// TIA Portal V19 export
FUNCTION_BLOCK "Sensors"   // FB4, LAD
{ S7_Optimized_Access := 'TRUE' }
// stored: MemoryReserve 100, SetENOAutomatically false
   VAR
      GenericSensor11 { S7_SetPoint := 'True'} : "GenericSensor";
      GenericSensor12 { S7_SetPoint := 'True'} : "GenericSensor";
      GenericSensor13 { S7_SetPoint := 'True'} : "GenericSensor";
      GenericSensor21 { S7_SetPoint := 'True'} : "GenericSensor";
      GenericSensor22 { S7_SetPoint := 'True'} : "GenericSensor";
      PubJsonMqttInst11 { S7_SetPoint := 'True'} : "PublishJsonMqtt";
      PubJsonMqttInst12 { S7_SetPoint := 'True'} : "PublishJsonMqtt";
      PubJsonMqttInst13 { S7_SetPoint := 'True'} : "PublishJsonMqtt";
      PubJsonMqttInst21 { S7_SetPoint := 'True'} : "PublishJsonMqtt";
      PubJsonMqttInst22 { S7_SetPoint := 'True'} : "PublishJsonMqtt";
      tpGen01 { S7_SetPoint := 'True'} : TP_TIME;
      tpGen02 { S7_SetPoint := 'True'} : TP_TIME;
      tpGen03 { S7_SetPoint := 'True'} : TP_TIME;
      tpGen04 { S7_SetPoint := 'True'} : TP_TIME;
   END_VAR
   VAR_TEMP
      Sensor11 : Real;
      Sensor12 : Real;
      Sensor13 : Real;
      Sensor21 : Real;
      Sensor22 : Real;
   END_VAR
   VAR_TEMP   // added for the SCL form of the ladder/FBD networks
      _w1 : Bool;
   END_VAR
BEGIN

REGION Network 1 (SCL): Generator for data publish Machine 1
   // Define how often sensors are polled and mqtt data sent.
   #tpGen01(IN:=NOT #tpGen02.Q,
            PT:=T#1S);

   #tpGen02(IN:=NOT #tpGen01.Q,
            PT:=T#50MS);
END_REGION

REGION Network 2 (SCL): Generator for data publish Machine 2
   #tpGen03(IN := NOT #tpGen04.Q,
            PT := T#3S);

   #tpGen04(IN := NOT #tpGen03.Q,
            PT := T#50MS);
END_REGION

REGION Network 3: Line 1 / Machine 1 / Sensor 001
   // SELECTOR defines if simulated sensor value or real IO-Link sensor value is evaluated and published by MQTT.
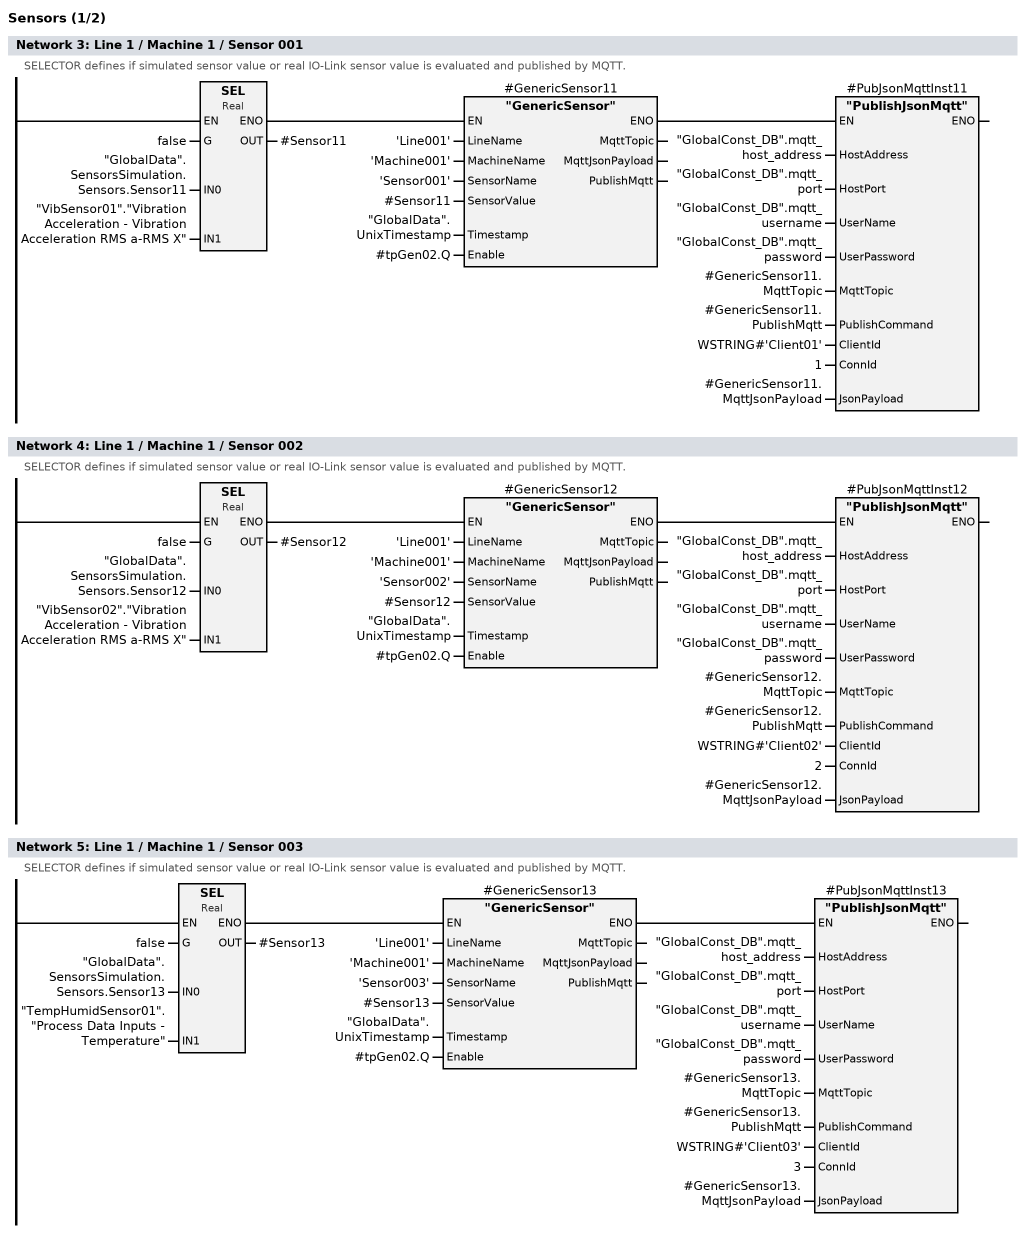
   RUNG wire#powerrail
      { S7_Templates := "value_type := Real" } SEL(g := false, in0 := "GlobalData".SensorsSimulation.Sensors.Sensor11, in1 := "VibSensor01"."Vibration Acceleration - Vibration Acceleration RMS a-RMS X", out => #Sensor11)
      #GenericSensor11(LineName := 'Line001', MachineName := 'Machine001', SensorName := 'Sensor001', SensorValue := #Sensor11, Timestamp := "GlobalData".UnixTimestamp, Enable := #tpGen02.Q, MqttTopic =>, MqttJsonPayload =>, PublishMqtt =>)
      #PubJsonMqttInst11(HostAddress := "GlobalConst_DB".mqtt_host_address, HostPort := "GlobalConst_DB".mqtt_port, UserName := "GlobalConst_DB".mqtt_username, UserPassword := "GlobalConst_DB".mqtt_password, MqttTopic := #GenericSensor11.MqttTopic, PublishCommand := #GenericSensor11.PublishMqtt, ClientId := WSTRING#'Client01', ConnId := 1, JsonPayload := #GenericSensor11.MqttJsonPayload)
   END_RUNG
   // the same network as SCL:
   // ENO of a box is taken as its EN; it also drops when the box reports an error
   #Sensor11 := SEL(G := false, IN0 := "GlobalData".SensorsSimulation.Sensors.Sensor11, IN1 := "VibSensor01"."Vibration Acceleration - Vibration Acceleration RMS a-RMS X");
   #GenericSensor11(LineName := 'Line001',   // "GenericSensor"
                    MachineName := 'Machine001',
                    SensorName := 'Sensor001',
                    SensorValue := #Sensor11,
                    Timestamp := "GlobalData".UnixTimestamp,
                    Enable := #tpGen02.Q,
                    ENO => #_w1);
   IF #_w1 THEN
       #PubJsonMqttInst11(HostAddress := "GlobalConst_DB".mqtt_host_address,   // "PublishJsonMqtt"
                          HostPort := "GlobalConst_DB".mqtt_port,
                          UserName := "GlobalConst_DB".mqtt_username,
                          UserPassword := "GlobalConst_DB".mqtt_password,
                          MqttTopic := #GenericSensor11.MqttTopic,
                          PublishCommand := #GenericSensor11.PublishMqtt,
                          ClientId := WSTRING#'Client01',
                          ConnId := 1,
                          JsonPayload := #GenericSensor11.MqttJsonPayload);
   END_IF;
END_REGION

REGION Network 4: Line 1 / Machine 1 / Sensor 002
   // SELECTOR defines if simulated sensor value or real IO-Link sensor value is evaluated and published by MQTT.
   RUNG wire#powerrail
      { S7_Templates := "value_type := Real" } SEL(g := false, in0 := "GlobalData".SensorsSimulation.Sensors.Sensor12, in1 := "VibSensor02"."Vibration Acceleration - Vibration Acceleration RMS a-RMS X", out => #Sensor12)
      #GenericSensor12(LineName := 'Line001', MachineName := 'Machine001', SensorName := 'Sensor002', SensorValue := #Sensor12, Timestamp := "GlobalData".UnixTimestamp, Enable := #tpGen02.Q, MqttTopic =>, MqttJsonPayload =>, PublishMqtt =>)
      #PubJsonMqttInst12(HostAddress := "GlobalConst_DB".mqtt_host_address, HostPort := "GlobalConst_DB".mqtt_port, UserName := "GlobalConst_DB".mqtt_username, UserPassword := "GlobalConst_DB".mqtt_password, MqttTopic := #GenericSensor12.MqttTopic, PublishCommand := #GenericSensor12.PublishMqtt, ClientId := WSTRING#'Client02', ConnId := 2, JsonPayload := #GenericSensor12.MqttJsonPayload)
   END_RUNG
   // the same network as SCL:
   // ENO of a box is taken as its EN; it also drops when the box reports an error
   #Sensor12 := SEL(G := false, IN0 := "GlobalData".SensorsSimulation.Sensors.Sensor12, IN1 := "VibSensor02"."Vibration Acceleration - Vibration Acceleration RMS a-RMS X");
   #GenericSensor12(LineName := 'Line001',   // "GenericSensor"
                    MachineName := 'Machine001',
                    SensorName := 'Sensor002',
                    SensorValue := #Sensor12,
                    Timestamp := "GlobalData".UnixTimestamp,
                    Enable := #tpGen02.Q,
                    ENO => #_w1);
   IF #_w1 THEN
       #PubJsonMqttInst12(HostAddress := "GlobalConst_DB".mqtt_host_address,   // "PublishJsonMqtt"
                          HostPort := "GlobalConst_DB".mqtt_port,
                          UserName := "GlobalConst_DB".mqtt_username,
                          UserPassword := "GlobalConst_DB".mqtt_password,
                          MqttTopic := #GenericSensor12.MqttTopic,
                          PublishCommand := #GenericSensor12.PublishMqtt,
                          ClientId := WSTRING#'Client02',
                          ConnId := 2,
                          JsonPayload := #GenericSensor12.MqttJsonPayload);
   END_IF;
END_REGION

REGION Network 5: Line 1 / Machine 1 / Sensor 003
   // SELECTOR defines if simulated sensor value or real IO-Link sensor value is evaluated and published by MQTT.
   RUNG wire#powerrail
      { S7_Templates := "value_type := Real" } SEL(g := false, in0 := "GlobalData".SensorsSimulation.Sensors.Sensor13, in1 := "TempHumidSensor01"."Process Data Inputs - Temperature", out => #Sensor13)
      #GenericSensor13(LineName := 'Line001', MachineName := 'Machine001', SensorName := 'Sensor003', SensorValue := #Sensor13, Timestamp := "GlobalData".UnixTimestamp, Enable := #tpGen02.Q, MqttTopic =>, MqttJsonPayload =>, PublishMqtt =>)
      #PubJsonMqttInst13(HostAddress := "GlobalConst_DB".mqtt_host_address, HostPort := "GlobalConst_DB".mqtt_port, UserName := "GlobalConst_DB".mqtt_username, UserPassword := "GlobalConst_DB".mqtt_password, MqttTopic := #GenericSensor13.MqttTopic, PublishCommand := #GenericSensor13.PublishMqtt, ClientId := WSTRING#'Client03', ConnId := 3, JsonPayload := #GenericSensor13.MqttJsonPayload)
   END_RUNG
   // the same network as SCL:
   // ENO of a box is taken as its EN; it also drops when the box reports an error
   #Sensor13 := SEL(G := false, IN0 := "GlobalData".SensorsSimulation.Sensors.Sensor13, IN1 := "TempHumidSensor01"."Process Data Inputs - Temperature");
   #GenericSensor13(LineName := 'Line001',   // "GenericSensor"
                    MachineName := 'Machine001',
                    SensorName := 'Sensor003',
                    SensorValue := #Sensor13,
                    Timestamp := "GlobalData".UnixTimestamp,
                    Enable := #tpGen02.Q,
                    ENO => #_w1);
   IF #_w1 THEN
       #PubJsonMqttInst13(HostAddress := "GlobalConst_DB".mqtt_host_address,   // "PublishJsonMqtt"
                          HostPort := "GlobalConst_DB".mqtt_port,
                          UserName := "GlobalConst_DB".mqtt_username,
                          UserPassword := "GlobalConst_DB".mqtt_password,
                          MqttTopic := #GenericSensor13.MqttTopic,
                          PublishCommand := #GenericSensor13.PublishMqtt,
                          ClientId := WSTRING#'Client03',
                          ConnId := 3,
                          JsonPayload := #GenericSensor13.MqttJsonPayload);
   END_IF;
END_REGION

REGION Network 6: Line 1 / Machine 2 / Sensor 001
   // SELECTOR defines if simulated sensor value or real IO-Link sensor value is evaluated and published by MQTT.
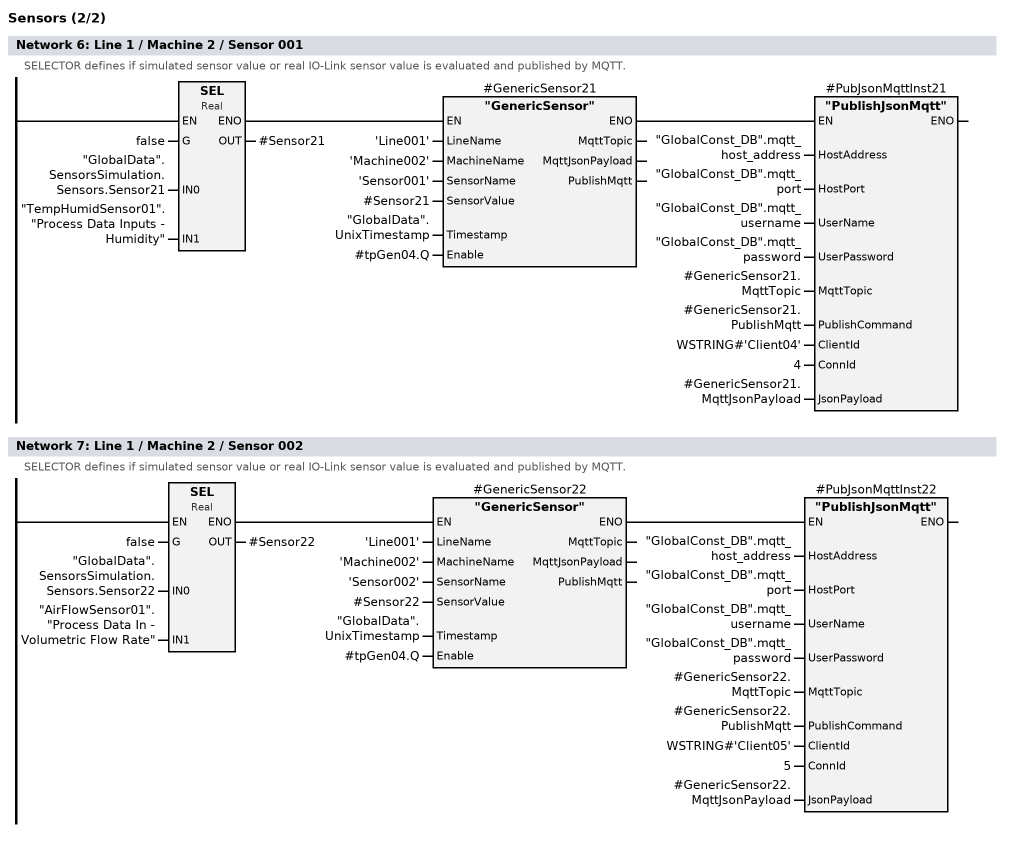
   RUNG wire#powerrail
      { S7_Templates := "value_type := Real" } SEL(g := false, in0 := "GlobalData".SensorsSimulation.Sensors.Sensor21, in1 := "TempHumidSensor01"."Process Data Inputs - Humidity", out => #Sensor21)
      #GenericSensor21(LineName := 'Line001', MachineName := 'Machine002', SensorName := 'Sensor001', SensorValue := #Sensor21, Timestamp := "GlobalData".UnixTimestamp, Enable := #tpGen04.Q, MqttTopic =>, MqttJsonPayload =>, PublishMqtt =>)
      #PubJsonMqttInst21(HostAddress := "GlobalConst_DB".mqtt_host_address, HostPort := "GlobalConst_DB".mqtt_port, UserName := "GlobalConst_DB".mqtt_username, UserPassword := "GlobalConst_DB".mqtt_password, MqttTopic := #GenericSensor21.MqttTopic, PublishCommand := #GenericSensor21.PublishMqtt, ClientId := WSTRING#'Client04', ConnId := 4, JsonPayload := #GenericSensor21.MqttJsonPayload)
   END_RUNG
   // the same network as SCL:
   // ENO of a box is taken as its EN; it also drops when the box reports an error
   #Sensor21 := SEL(G := false, IN0 := "GlobalData".SensorsSimulation.Sensors.Sensor21, IN1 := "TempHumidSensor01"."Process Data Inputs - Humidity");
   #GenericSensor21(LineName := 'Line001',   // "GenericSensor"
                    MachineName := 'Machine002',
                    SensorName := 'Sensor001',
                    SensorValue := #Sensor21,
                    Timestamp := "GlobalData".UnixTimestamp,
                    Enable := #tpGen04.Q,
                    ENO => #_w1);
   IF #_w1 THEN
       #PubJsonMqttInst21(HostAddress := "GlobalConst_DB".mqtt_host_address,   // "PublishJsonMqtt"
                          HostPort := "GlobalConst_DB".mqtt_port,
                          UserName := "GlobalConst_DB".mqtt_username,
                          UserPassword := "GlobalConst_DB".mqtt_password,
                          MqttTopic := #GenericSensor21.MqttTopic,
                          PublishCommand := #GenericSensor21.PublishMqtt,
                          ClientId := WSTRING#'Client04',
                          ConnId := 4,
                          JsonPayload := #GenericSensor21.MqttJsonPayload);
   END_IF;
END_REGION

REGION Network 7: Line 1 / Machine 2 / Sensor 002
   // SELECTOR defines if simulated sensor value or real IO-Link sensor value is evaluated and published by MQTT.
   RUNG wire#powerrail
      { S7_Templates := "value_type := Real" } SEL(g := false, in0 := "GlobalData".SensorsSimulation.Sensors.Sensor22, in1 := "AirFlowSensor01"."Process Data In - Volumetric Flow Rate", out => #Sensor22)
      #GenericSensor22(LineName := 'Line001', MachineName := 'Machine002', SensorName := 'Sensor002', SensorValue := #Sensor22, Timestamp := "GlobalData".UnixTimestamp, Enable := #tpGen04.Q, MqttTopic =>, MqttJsonPayload =>, PublishMqtt =>)
      #PubJsonMqttInst22(HostAddress := "GlobalConst_DB".mqtt_host_address, HostPort := "GlobalConst_DB".mqtt_port, UserName := "GlobalConst_DB".mqtt_username, UserPassword := "GlobalConst_DB".mqtt_password, MqttTopic := #GenericSensor22.MqttTopic, PublishCommand := #GenericSensor22.PublishMqtt, ClientId := WSTRING#'Client05', ConnId := 5, JsonPayload := #GenericSensor22.MqttJsonPayload)
   END_RUNG
   // the same network as SCL:
   // ENO of a box is taken as its EN; it also drops when the box reports an error
   #Sensor22 := SEL(G := false, IN0 := "GlobalData".SensorsSimulation.Sensors.Sensor22, IN1 := "AirFlowSensor01"."Process Data In - Volumetric Flow Rate");
   #GenericSensor22(LineName := 'Line001',   // "GenericSensor"
                    MachineName := 'Machine002',
                    SensorName := 'Sensor002',
                    SensorValue := #Sensor22,
                    Timestamp := "GlobalData".UnixTimestamp,
                    Enable := #tpGen04.Q,
                    ENO => #_w1);
   IF #_w1 THEN
       #PubJsonMqttInst22(HostAddress := "GlobalConst_DB".mqtt_host_address,   // "PublishJsonMqtt"
                          HostPort := "GlobalConst_DB".mqtt_port,
                          UserName := "GlobalConst_DB".mqtt_username,
                          UserPassword := "GlobalConst_DB".mqtt_password,
                          MqttTopic := #GenericSensor22.MqttTopic,
                          PublishCommand := #GenericSensor22.PublishMqtt,
                          ClientId := WSTRING#'Client05',
                          ConnId := 5,
                          JsonPayload := #GenericSensor22.MqttJsonPayload);
   END_IF;
END_REGION
END_FUNCTION_BLOCK
